{attribute 'linkalways'} 
{attribute 'no_explicit_call' := 'This FB is a CLASS and must be accessed using methods or properties'}
{attribute 'enable_dynamic_creation'}
FUNCTION_BLOCK Node_F_VN_InsertIntoContainer_LREAL EXTENDS VisionNode
VAR
    fElement : _LREAL(0.0);
    ipContainer : _ITcVnContainer;
    nIndex : _ULINT(0);
    hrPrev : _HRESULT(S_OK);
    hresult : _HRESULT(S_OK);
END_VAR

METHOD PUBLIC  Clone : I_Node
VAR
	pNode : POINTER TO Node_F_VN_InsertIntoContainer_LREAL;
END_VAR
pNode := __NEW(Node_F_VN_InsertIntoContainer_LREAL);
Clone := pNode^;
END_METHOD

METHOD FB_init : BOOL
VAR_INPUT
	bInitRetains : BOOL; // if TRUE, the retain variables are initialized (warm start / cold start)
	bInCopyCode : BOOL;  // if TRUE, the instance afterwards gets moved into the copy code (online change)
END_VAR
AddInput('fElement', fElement);
AddInput('ipContainer', ipContainer);
AddInput('nIndex', nIndex);
AddInput('hrPrev', hrPrev);
AddOutput('ipContainer', ipContainer);
AddOutput('hresult',hresult);
END_METHOD

METHOD PROTECTED OnExecute : HRESULT
hresult.Value := F_VN_InsertIntoContainer_LREAL(
    fElement := fElement.Value,
    ipContainer := ipContainer.Value,
    nIndex := nIndex.Value,
    hrPrev:= hrPrev.Value);
END_METHOD

METHOD PUBLIC PreExecutionCheck
VAR_INPUT
	Check : I_PreExecutionChecks;
END_VAR
Check.IsTrue(ipContainer.IsValid, 'ipContainer must be a valid container');
END_METHOD

END_FUNCTION_BLOCK

(* stored: Version 1.1.0.1, ProductVersion 3.1.4024.13
   POU Node_F_VN_InsertIntoContainer_LREAL: Id {2e1a0409-432e-429a-95a6-d8527819d9d0}, SpecialFunc None
   Folder Constructor: Id {28d96288-4855-4bbd-b395-a02b58f1f7d9}
   Method Clone: Id {61b61337-b025-472f-b911-ae2f3f71ee0d}
   Method FB_init: Id {9c25adc4-1f67-455f-8680-1eaf671842f3}
   Method OnExecute: Id {7da37536-efe5-4022-a7df-f2d4452ce6c0}
   Method PreExecutionCheck: Id {97491edb-8c85-4564-b92c-154e7a9c7dd2} *)
